// TIA Portal V18 export
DATA_BLOCK "DataLogging_DB"   // DB94
VERSION : 0.1
// stored: AutoNumber true, DBAccessibleFromOPCUA true, InstanceOfName DataLogging, InstanceOfType FB
"DataLogging"
   // VAR_INPUT
   //    CreateFile : Bool;
   //    StartLogging : Bool;
   //    Variable01in_Bool : Bool;
   //    Name_01 : String;
   //    Variable02in_Bool : Bool;
   //    Name_02 : String;
   //    Variable03in_Dint : DInt;
   //    Name_03 : String;
   //    Variable04in_Dint : DInt;
   //    Name_04 : String;
   //    Variable05in_Dint : DInt;
   //    Name_05 : String;
   //    Variable06in_Dint : DInt;
   //    Name_06 : String;
   // END_VAR
   // VAR_OUTPUT
   //    Variable01out_Bool : Bool;
   //    Variable02out_Bool : Bool;
   //    Variable03out_Dint : DInt;
   //    Variable04out_Dint : DInt;
   //    Variable05out_Dint : DInt;
   //    Variable06out_Dint : DInt;
   //    LogColumns : String;
   // END_VAR
   // VAR
   //    FileName : String;
   //    REQ : Bool;
   //    ID : DWord;
   //    StartingTime : DTL;
   //    ReturnValue : Int;
   //    AmountOfRecords : UDInt;
   //    StartLoggingM : Bool;
   //    WriteColumn : Int;
   //    Column01Internal { ExternalAccessible := 'False'; ExternalVisible := 'False'; ExternalWritable := 'False'} : String;
   //    Column02Internal { ExternalAccessible := 'False'; ExternalVisible := 'False'; ExternalWritable := 'False'} : String;
   //    Column03Internal { ExternalAccessible := 'False'; ExternalVisible := 'False'; ExternalWritable := 'False'} : String;
   //    Column04Internal { ExternalAccessible := 'False'; ExternalVisible := 'False'; ExternalWritable := 'False'} : String;
   //    Column05Internal : String;
   //    Column06Internal : String;
   //    WriteColumnReady : Bool;
   //    RecordCount : DInt;
   // END_VAR
BEGIN
END_DATA_BLOCK
